(* IEC 61131-3 sources: programs/VI-54/VI-54_20171205/VI-54_20171205/Stations/Screen/LseClass170718/Class/DiagnosticStationBase, 1 file *)

(* ---- DiagnosticStationBase.st ---- *)
(*!
<Class
	Name               = "DiagnosticStationBase"
	Revision           = "1.0"
	RealtimeTask       = "false"
	CyclicTask         = "false"
	BackgroundTask     = "true"
	Sigmatek           = "false"
	OSInterface        = "false"
	HighPriority       = "false"
	Automatic          = "false"
	UpdateMode         = "Prescan"
	SharedCommandTable = "true"
	Objectsize         = "(438,120)"
	Comment            = "Use this class as base class for new stations.">
	<Channels>
		<Server Name="sStationName" Class="StringInternal" Visualized="true" Remotely="true" Initialize="true" WriteProtected="false" Retentive="false" Comment="Name of the station."/>
		<Server Name="sStatus" Visualized="false" Initialize="false" WriteProtected="true" Retentive="false" Comment="Actual state of the station."/>
		<Client Name="cHandler" Required="true" Internal="false" Comment="Object channel to DiagnosticStationHandlerBase."/>
		<Client Name="cSigCLib" Required="false" Internal="false" Comment="Object channel to SigCLib. Does not have to be connected."/>
		<Client Name="StationName" Required="true" Internal="true"/>
	</Channels>
	<RevDoku>
		<Owner Company="Sigmatek"/>
		<Dokumentation Revision="1.0" Date="2016-06-02" Author="HötAnt" Company="Sigmatek" Description="Creation"/>
	</RevDoku>
	<Network Name="DiagnosticStationBase">
		<!-- List of Components in this network -->
		<Components>
			<Object
				Name       = "StationName"
				Class      = "String"
				Position   = "(150,300)"
				Visualized = "true"
				Remotely   = "true">
				<Channels>
					<Server Name="Data"/>
					<Client Name="SingleRealloc" Value="1"/>
				</Channels>
			</Object>
		</Components>
		<Comments>
		</Comments>
		<!-- List of Connections in this network -->
		<Connections>
			<Connection Source="this.StationName" Destination="StationName.Data"/>
			<Connection Source="this.sStationName" Destination="StationName.Data" Vertices="(878,270),(706,390),"/>
		</Connections>
		<!-- Headerfiles -->
		<Options>
		</Options>
	</Network>
</Class>
*)
DiagnosticStationBase : CLASS
  //Servers:
	sStatus 	: SvrChCmd_iprStates;
	sStationName 	: SvrChCmd_UDINT;
  //Clients:
	cHandler 	: CltChCmd_DiagnosticStationHandlerBase;
	StationName 	: CltChCmd_String;
	cSigCLib 	: CltChCmd_SigCLib;
  //Variables:
		NameOfStation 	: _DiagString;
  //Functions:

	FUNCTION VIRTUAL GLOBAL Init;

	FUNCTION VIRTUAL GLOBAL Background
		VAR_INPUT
			EAX 	: UDINT;
		END_VAR
		VAR_OUTPUT
			state (EAX) 	: UDINT;
		END_VAR;
				//! <Function Comment="This method is called when the diagnostic export starts. Overwrite it to react to the start of the diagnostic export." Name="StartAction"/>
	FUNCTION VIRTUAL GLOBAL StartAction
		VAR_INPUT
			pDP 	: ^CHAR;			//! <Variable Comment="Pointer to the folder path." Name="StartAction.pDP"/>
		END_VAR
		VAR_OUTPUT
			retcode 	: BOOL;			//! <Variable Comment="FALSE..Error&#13;&#10;TRUE..Ok" Name="StartAction.retcode"/>
		END_VAR;
				//! <Function Comment="This method returns the actual state of the station." Name="GetWorkState"/>
	FUNCTION VIRTUAL GLOBAL GetWorkState
		VAR_OUTPUT
			retcode 	: iprStates;			//! <Variable Comment="Actual status." Name="GetWorkState.retcode"/>
		END_VAR;
				//! <Function Comment="This method returns the name of the station." Name="GetStationName"/>
	FUNCTION VIRTUAL GetStationName
		VAR_OUTPUT
			pName 	: ^CHAR;			//! <Variable Comment="Pointer to the station name." Name="GetStationName.pName"/>
		END_VAR;
				//! <Function Comment="Call the method SetError from the DiagnosticStationHandlerBase class with your error number and your error code." Name="SetError"/>
	FUNCTION GLOBAL SetError
		VAR_INPUT
			ErrorNr 	: DINT;			//! <Variable Comment="Error number." Name="SetError.ErrorNr"/>
			ErrorCode 	: DINT;			//! <Variable Comment="Error code." Name="SetError.ErrorCode"/>
		END_VAR;
  //Tables:
	FUNCTION @STD
		VAR_OUTPUT
			ret_code	: CONFSTATES;
		END_VAR;
	FUNCTION GLOBAL TAB @CT_;
END_CLASS;

#pragma using String
#pragma usingLtd DiagnosticStationHandlerBase
#pragma usingLtd SigCLib

// ********************************************************************
// Prototype of StartAction Methode
// ********************************************************************
// ********************************************************************
#pragma warning(disable:73);

FUNCTION GLOBAL PT_STARTACTION_FNC_DiagnosticStationBase
	VAR_INPUT
		pthis 	: ^void;
    pDP     : ^char;
	END_VAR
  var_output
    retcode : dint;
  end_var

  retcode := pthis$^DiagnosticStationBase^.StartAction(pDP);

END_FUNCTION

FUNCTION VIRTUAL GLOBAL DiagnosticStationBase::StartAction
	VAR_INPUT
		pDP 	: ^CHAR;
	END_VAR
	VAR_OUTPUT
		retcode 	: BOOL;
	END_VAR

  retcode := TRUE;
  sStatus := BUSY;

END_FUNCTION
#pragma warning(default:73);
// ********************************************************************
// Prototype of GetWorkState Methode
// ********************************************************************
// ********************************************************************
FUNCTION GLOBAL PT_GETSTATE_FNC_DiagnosticStationBase
	VAR_INPUT
		pthis 	: ^void;
	END_VAR
  var_output
    retcode : iprStates;
  end_var

  retcode := pthis$^DiagnosticStationBase^.GetWorkState();

END_FUNCTION

FUNCTION VIRTUAL GLOBAL DiagnosticStationBase::GetWorkState
	VAR_OUTPUT
		retcode 	: iprStates;
	END_VAR

  retcode := sstatus;

END_FUNCTION

FUNCTION VIRTUAL GLOBAL DiagnosticStationBase::Init

  if _FirstScan then
    // Station meldet sich bei der Funktion an , um im Falle eines Export aufgerufen zu werden.
    cHandler.InstallStation(pname:= GetStationName(),
                            pThis:=this,
                            pFct_StartAction:=#PT_STARTACTION_FNC_DiagnosticStationBase(),
                            pFct_GetState:=#PT_GETSTATE_FNC_DiagnosticStationBase());
  end_if;

END_FUNCTION

FUNCTION VIRTUAL GLOBAL DiagnosticStationBase::Background
	VAR_INPUT
		EAX 	: UDINT;
	END_VAR
	VAR_OUTPUT
		state (EAX) 	: UDINT;
	END_VAR

	state := READY;

END_FUNCTION

FUNCTION VIRTUAL DiagnosticStationBase::GetStationName
	VAR_OUTPUT
		pName 	: ^CHAR;
	END_VAR

  StationName.ReadDataOff(udOff:=0, pData:=#NameOfStation[0], udMax:=sizeof(NameOfStation));
  pName := #NameOfStation[0];

END_FUNCTION

FUNCTION GLOBAL DiagnosticStationBase::SetError
	VAR_INPUT
		ErrorNr 	: DINT;
		ErrorCode 	: DINT;
	END_VAR

  cHandler.SetError(pStationName:=GetStationName(), ErrorNr, ErrorCode);

END_FUNCTION
